(* CoDeSys 2.3.9.47 project: bmwWrote.pro *)
(* Libraries: WagoCANLayer2_02.lib 23.6.14 12:08:28, Standard.lib 20.5.14 07:13:26, Iecsfc.lib 16.5.13 13:00:50, SYSLIBCALLBACK.LIB 16.5.13 13:00:50 *)

(* PLC configuration (modules and I/O channels)
K-Bus [K_Bus] node 0, in %IB0 out %QB0 {KbusBusMode = 1; KbusCycleTime = 10000; KbusThreadPriority = 0; KbusSetOutputsToZeroOnApplicationStop = 1}
Modbus variables [PFC200MODBUS] node 1, in %IB0 out %QB0 {PlcStopBehaviour = 1; FiledbusErrorBehaviour = 1; TcpOperation = 1; TcpPort = 502; TcpTimeout = 600; UdpOperation = 1; UdpPort = 502; RtuOperation = 0; NodeId = 1; ResponseTimeout = 5000; Interface = 0; Baud = 115200; StopBits = 1; Parity = 1; FlowCtrl = 0; PhysInterface = 0}
CAN Layer2 Device [PFC200CANLAYER2] node 2, in %IB6000 out %QB6000 {PFC200CanLayer2NONE = 0}
Modbus-Master [MB_MASTER] node 3, in %IB0 out %QB0
*)

(* Task configuration *)
TASK T500 (PRIORITY := 31, INTERVAL := T#100ms);
	PLC_PRG();
END_TASK

(* POU PLC_PRG, ST *)
PROGRAM PLC_PRG
VAR
	xOpenPort			: BOOL;
	fbOpenPort		: CAN_OPEN;
	xPortIsOpen		: BOOL;
	fbCanSend1			: CAN_TX_11BIT_FRAME :=(
		CAN_ID			:= 16#0351,
		RTR_FRAME		:= FALSE,
		DATALENGTH	:= 8 );
	fbCanSend2			: CAN_TX_11BIT_FRAME :=(
		CAN_ID			:= 16#0355,
		RTR_FRAME		:= FALSE,
		DATALENGTH	:= 8 );
	fbCanSend3		: CAN_TX_11BIT_FRAME :=(
		CAN_ID			:= 16#0356,
		RTR_FRAME		:= FALSE,
		DATALENGTH	:= 8 );
	fbCanSendAlarms		: CAN_TX_11BIT_FRAME :=(
		CAN_ID			:= 16#035A,
		RTR_FRAME		:= FALSE,
		DATALENGTH	:= 8 );

	fbCanRecv1			: CAN_RX_11BIT_FRAME :=(
		CAN_ID			:= 16#0305,
		CAN_BUFFER	:= FALSE );
	fbCanRecv2			: CAN_RX_11BIT_FRAME :=(
		CAN_ID			:= 16#0306,
		CAN_BUFFER	:= FALSE );
	fbCanRecv3			: CAN_RX_11BIT_FRAME :=(
		CAN_ID			:= 16#0307,
		CAN_BUFFER	:= FALSE );

	xWrite					: BOOL;
	xRead					: BOOL;
	wState					: WORD;

	aSendData1			: ARRAY [1..8] OF BYTE; (* :=80, 0, 0, 0, 0, 0, 0, 0;*)
	aSendData2			: ARRAY [1..8] OF BYTE;
	aSendData3			: ARRAY [1..8] OF BYTE :=  87, 20, 254, 255, 199, 0, 0 , 0;
	aSendData4			: ARRAY [1..8] OF BYTE  := 170, 170, 170, 170, 170, 170, 170,  170;

	aRecvData1			: ARRAY [1..8] OF BYTE;
	aRecvData2			: ARRAY [1..8] OF BYTE;
	aRecvData3			: ARRAY [1..8] OF BYTE;
	bRecvLen				: BYTE;
	tSend					: TON :=(PT:= t#10ms );
END_VAR
fbOpenPort(BAUDRATE:= 500000, ENABLE:= xOpenPort);

fbCanRecv1(
	ENABLE:= xPortIsOpen,
	READ_FRAME:= xRead );

fbCanRecv2(
	ENABLE:= xPortIsOpen,
	READ_FRAME:= xRead );

fbCanRecv3(
	ENABLE:= xPortIsOpen,
	READ_FRAME:= xRead );


fbCanSend1(
	DATA:= aSendData1,
	ENABLE:= xPortIsOpen,
	WRITE_FRAME:= xWrite );


fbCanSend2(
	DATA:= aSendData2,
	ENABLE:= xPortIsOpen,
	WRITE_FRAME:= xWrite );


fbCanSend3(
	DATA:= aSendData3,
	ENABLE:= xPortIsOpen,
	WRITE_FRAME:= xWrite );

fbCanSendAlarms(
	DATA:= aSendData4,
	ENABLE:= xPortIsOpen,
	WRITE_FRAME:= xWrite );


CASE wState OF
0: (* open CAN port *)
	xOpenPort := TRUE;
	IF fbOpenPort.CONFIRM AND fbOpenPort.ERROR = CAN_PORT_OK THEN
		xOpenPort := FALSE;
		xPortIsOpen := TRUE;
		wState := 10;
	END_IF
10: (* send cyclic messages and check if message was received *)
	tSend(IN := TRUE AND NOT xWrite);
	IF tSend.Q THEN (* sending message *)
		tSend(IN := FALSE);
		xWrite := TRUE;
	ELSIF NOT xRead THEN (* message received *)
		IF fbCanRecv1.ERROR = CAN_RECEIVE_OK OR  fbCanRecv2.ERROR = CAN_RECEIVE_OK OR  fbCanRecv3.ERROR = CAN_RECEIVE_OK THEN
			aRecvData1 := fbCanRecv1.DATA;
			aRecvData2 := fbCanRecv2.DATA;
			aRecvData3 := fbCanRecv3.DATA;

			(*16#305 -> 16#351*)
			aSendData1[1] := 103; (*aRecvData1[0];*)
			aSendData1[2] := 2;     (*aRecvData1[1]*)
			aSendData1[3] := 52;
			aSendData1[4] := 3;
			aSendData1[5] := 126;
			aSendData1[6] := 9;
			aSendData1[7] := 164;
			aSendData1[8] := 1;

			(*16#306 -> 16#355*)
			aSendData2[1] := aRecvData1[7];
			aSendData2[2] := aRecvData1[8];
			aSendData2[3] := aRecvData2[1];
			aSendData2[4] := aRecvData2[2];
			aSendData2[5] := 140;
			aSendData2[6] := 10;
			aSendData2[7] := 0;
			aSendData2[8] := 0;

			(*16#306 -> 16#356*)
			(*aSendData3 := 87, 20, 254, 255, 199, 0, 0 , 0;*)

			bRecvLen := fbCanRecv1.DATALENGTH;
			xRead := TRUE;
		ELSE
			xRead := TRUE;
		END_IF
	END_IF
END_CASE
END_PROGRAM
